FUNCTION_BLOCK AX_R_TRIG (* Boolean rising edge detection *)
  (* Standard: 61499-1 Annex A; Description: Copyright (c) 2017 fortiss GmbH, HR Agrartechnik GmbH This program and the accompanying materials are made available under the terms of the Eclipse Public License 2.0 which is available at https://www.eclipse.org/legal/epl-2.0/ SPDX-License-Identifier: EPL-2.0 *)
  (* Version 3.0, 2025-04-14, Patrick Aigner, changed package *)
  (* Version 1.0, 2017-09-22, Alois Zoitl, fortiss GmbH, initial API and implementation and/or initial documentation *)
  PACKAGE adapter::events::unidirectional;
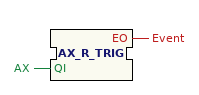
  EVENT_OUTPUT
    EO; (* confirmation that an rising edge was detected *)
  END_EVENT
  SOCKETS
    QI : adapter::types::unidirectional::AX; (* value to check for a rising edge *)
  END_SOCKETS
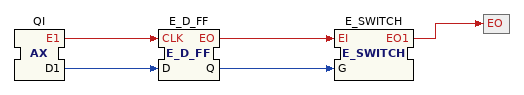
  FBS
    E_D_FF : iec61499::events::E_D_FF;
    E_SWITCH : iec61499::events::E_SWITCH;
  END_FBS
  EVENT_CONNECTIONS
    E_D_FF.EO TO E_SWITCH.EI;
    E_SWITCH.EO1 TO EO;
    QI.E1 TO E_D_FF.CLK;
  END_CONNECTIONS
  DATA_CONNECTIONS
    E_D_FF.Q TO E_SWITCH.G;
    QI.D1 TO E_D_FF.D;
  END_CONNECTIONS
END_FUNCTION_BLOCK
